Yaskawa INFORM job: kufsa_test_with_table.JBI

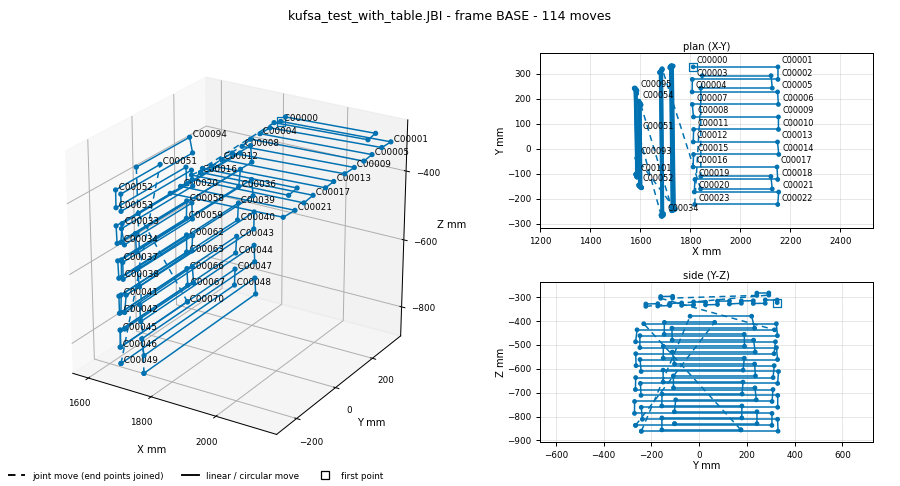
[picture p0: tool path of kufsa_test_with_table.JBI in frame BASE, 114 of 114 moves have a stored position in this frame; points joined in program order, loops and branches not executed]
/JOB
//NAME kufsa_with_table
//POS
///NPOS 114,0,114,0,0,0
///TOOL 0
///POSTYPE BASE
///RECTAN
///RCONF 1,0,0,0,0,0,0,0,0,0,0,0,0,0,0,0,0,0,0,0,0,0,0,0
C00000=1812.070007,326.956462,-322.467041,180.000000,-89.999999,0.000000
C00001=2150.695598,326.956462,-312.028718,180.000000,-89.999999,0.000000
C00002=2150.727599,276.956462,-311.505303,180.000000,-89.999999,0.000000
C00003=1808.470333,276.956462,-325.644002,180.000000,-89.999999,0.000000
C00004=1807.754534,226.956462,-326.266171,180.000000,-89.999999,0.000000
C00005=2149.229584,226.956462,-314.850962,180.000000,-89.999999,0.000000
C00006=2152.427886,176.956462,-315.522758,180.000000,-89.999999,0.000000
C00007=1808.354706,176.956462,-325.499784,180.000000,-89.999999,0.000000
C00008=1813.127705,126.956462,-328.391472,180.000000,-89.999999,0.000000
C00009=2152.547136,126.956462,-316.102628,180.000000,-89.999999,0.000000
C00010=2152.688424,76.956462,-316.428035,180.000000,-89.999999,0.000000
C00011=1813.792182,76.956462,-330.537424,180.000000,-89.999999,0.000000
C00012=1812.079517,26.956462,-332.110167,180.000000,-89.999999,0.000000
C00013=2148.963612,26.956462,-320.940761,180.000000,-89.999999,0.000000
C00014=2153.965148,-23.043538,-319.751379,180.000000,-89.999999,0.000000
C00015=1813.274428,-23.043538,-332.397937,180.000000,-89.999999,0.000000
C00016=1811.443268,-73.043538,-334.200996,180.000000,-89.999999,0.000000
C00017=2146.917653,-73.043538,-323.945193,180.000000,-89.999999,0.000000
C00018=2149.737979,-123.043538,-326.004047,180.000000,-89.999999,0.000000
C00019=1819.062406,-123.043538,-334.939239,180.000000,-89.999999,0.000000
C00020=1816.212947,-173.043538,-337.150638,180.000000,-89.999999,0.000000
C00021=2153.683780,-173.043538,-327.184770,180.000000,-89.999999,0.000000
C00022=2149.816473,-223.043538,-328.439434,180.000000,-89.999999,0.000000
C00023=1817.967726,-223.043538,-338.250259,180.000000,-89.999999,0.000000
C00024=1847.834252,291.859988,-291.167343,180.000000,-89.999999,0.000000
C00025=2123.193751,291.859988,-282.202509,180.000000,-89.999999,0.000000
C00026=2127.968562,241.859988,-282.721095,180.000000,-89.999999,0.000000
C00027=1842.147711,241.859988,-292.609524,180.000000,-89.999999,0.000000
C00028=1842.355615,-110.851952,-303.697098,180.000000,-89.999999,0.000000
C00029=2122.511360,-110.851952,-296.331318,180.000000,-89.999999,0.000000
C00030=2127.898871,-160.851952,-297.180806,180.000000,-89.999999,0.000000
C00031=1841.572191,-160.851952,-304.679312,180.000000,-89.999999,0.000000
C00032=1689.025256,316.314359,-436.599221,180.000000,-89.999999,0.000000
C00033=1693.340579,-259.742111,-436.599221,180.000000,-89.999999,0.000000
C00034=1692.565910,-265.923822,-486.599221,180.000000,-89.999999,0.000000
C00035=1687.558336,319.676130,-486.599221,180.000000,-89.999999,0.000000
C00036=1685.839030,313.772706,-536.599221,180.000000,-89.999999,0.000000
C00037=1691.883319,-265.207335,-536.599221,180.000000,-89.999999,0.000000
C00038=1690.585462,-264.079002,-586.599221,180.000000,-89.999999,0.000000
C00039=1684.578004,314.403429,-586.599221,180.000000,-89.999999,0.000000
C00040=1684.322900,309.849895,-636.599221,180.000000,-89.999999,0.000000
C00041=1689.091070,-265.469540,-636.599221,180.000000,-89.999999,0.000000
C00042=1687.752456,-266.658623,-686.599221,180.000000,-89.999999,0.000000
C00043=1681.655032,309.368812,-686.599221,180.000000,-89.999999,0.000000
C00044=1680.951913,305.521491,-736.599221,180.000000,-89.999999,0.000000
C00045=1687.427916,-270.100352,-736.599221,180.000000,-89.999999,0.000000
C00046=1685.190554,-270.446758,-786.599221,180.000000,-89.999999,0.000000
C00047=1678.938861,305.219084,-786.599221,180.000000,-89.999999,0.000000
C00048=1677.146797,304.775970,-836.599221,180.000000,-89.999999,0.000000
C00049=1683.692237,-266.007352,-836.599221,180.000000,-89.999999,0.000000
C00050=1683.692237,-266.007352,-836.599221,180.000000,-89.999999,0.000000
C00051=1592.682564,65.013086,-405.440930,180.000000,-89.999999,0.000000
C00052=1593.996273,-145.301390,-405.440930,180.000000,-89.999999,0.000000
C00053=1594.466635,-146.306407,-455.440930,180.000000,-89.999999,0.000000
C00054=1593.576386,188.991519,-455.440930,180.000000,-89.999999,0.000000
C00055=1594.547485,190.175259,-505.440930,180.000000,-89.999999,0.000000
C00056=1596.012621,-149.877854,-505.440930,180.000000,-89.999999,0.000000
C00057=1598.057111,-150.260962,-555.440930,180.000000,-89.999999,0.000000
C00058=1594.819072,189.154091,-555.440930,180.000000,-89.999999,0.000000
C00059=1596.462882,184.159348,-605.440930,180.000000,-89.999999,0.000000
C00060=1599.097893,-150.679694,-605.440930,180.000000,-89.999999,0.000000
C00061=1601.194645,-150.579766,-655.440930,180.000000,-89.999999,0.000000
C00062=1596.716601,183.692011,-655.440930,180.000000,-89.999999,0.000000
C00063=1598.777618,180.083430,-705.440930,180.000000,-89.999999,0.000000
C00064=1603.311051,-155.279706,-705.440930,180.000000,-89.999999,0.000000
C00065=1604.512194,-156.238230,-755.440930,180.000000,-89.999999,0.000000
C00066=1599.772168,179.164152,-755.440930,180.000000,-89.999999,0.000000
C00067=1602.114821,178.707079,-805.440930,180.000000,-89.999999,0.000000
C00068=1604.713204,-155.716551,-805.440930,180.000000,-89.999999,0.000000
C00069=1606.157345,-155.900105,-855.440930,180.000000,-89.999999,0.000000
C00070=1603.002390,174.947550,-855.440930,180.000000,-89.999999,0.000000
C00071=1603.002390,174.947550,-855.440930,180.000000,-89.999999,0.000000
C00072=1724.578416,-231.807524,-411.083672,180.000000,-89.999999,0.000000
C00073=1718.279325,323.447595,-411.083672,180.000000,-89.999999,0.000000
C00074=1719.725414,327.955120,-461.083672,180.000000,-89.999999,0.000000
C00075=1725.796875,-247.885600,-461.083672,180.000000,-89.999999,0.000000
C00076=1727.476934,-248.031667,-511.083672,180.000000,-89.999999,0.000000
C00077=1721.770468,323.709354,-511.083672,180.000000,-89.999999,0.000000
C00078=1723.614458,328.610857,-561.083672,180.000000,-89.999999,0.000000
C00079=1728.674863,-247.324114,-561.083672,180.000000,-89.999999,0.000000
C00080=1731.265446,-242.598605,-611.083672,180.000000,-89.999999,0.000000
C00081=1724.878351,332.404799,-611.083672,180.000000,-89.999999,0.000000
C00082=1725.967145,328.907011,-661.083672,180.000000,-89.999999,0.000000
C00083=1733.123323,-245.670029,-661.083672,180.000000,-89.999999,0.000000
C00084=1733.584924,-243.188232,-711.083672,180.000000,-89.999999,0.000000
C00085=1726.804307,329.270615,-711.083672,180.000000,-89.999999,0.000000
C00086=1729.229751,328.994115,-761.083672,180.000000,-89.999999,0.000000
C00087=1734.901952,-242.222270,-761.083672,180.000000,-89.999999,0.000000
C00088=1737.913833,-237.463930,-811.083672,180.000000,-89.999999,0.000000
C00089=1730.236277,328.580483,-811.083672,180.000000,-89.999999,0.000000
C00090=1731.867128,330.516874,-861.083672,180.000000,-89.999999,0.000000
C00091=1739.462265,-241.828515,-861.083672,180.000000,-89.999999,0.000000
C00092=1739.462265,-241.828515,-861.083672,180.000000,-89.999999,0.000000
C00093=1586.192316,-37.777443,-379.657788,180.000000,-89.999999,0.000000
C00094=1586.018778,220.048604,-379.657788,180.000000,-89.999999,0.000000
C00095=1587.115619,232.433194,-429.657788,180.000000,-89.999999,0.000000
C00096=1587.946012,-113.769722,-429.657788,180.000000,-89.999999,0.000000
C00097=1586.574680,-112.699043,-479.657788,180.000000,-89.999999,0.000000
C00098=1585.601795,228.117871,-479.657788,180.000000,-89.999999,0.000000
C00099=1584.980452,234.981511,-529.657788,180.000000,-89.999999,0.000000
C00100=1586.351337,-112.328011,-529.657788,180.000000,-89.999999,0.000000
C00101=1587.981300,-102.830919,-579.657788,180.000000,-89.999999,0.000000
C00102=1583.294206,232.360436,-579.657788,180.000000,-89.999999,0.000000
C00103=1582.141752,235.917997,-629.657788,180.000000,-89.999999,0.000000
C00104=1584.825898,-107.857211,-629.657788,180.000000,-89.999999,0.000000
C00105=1584.372957,-107.195150,-679.657788,180.000000,-89.999999,0.000000
C00106=1583.512190,233.854829,-679.657788,180.000000,-89.999999,0.000000
C00107=1577.236228,239.550729,-729.657788,180.000000,-89.999999,0.000000
C00108=1586.464349,-97.948331,-729.657788,180.000000,-89.999999,0.000000
C00109=1584.137106,-103.589890,-779.657788,180.000000,-89.999999,0.000000
C00110=1576.249941,242.210446,-779.657788,180.000000,-89.999999,0.000000
C00111=1580.180793,242.276562,-829.657788,180.000000,-89.999999,0.000000
C00112=1582.279332,-102.714387,-829.657788,180.000000,-89.999999,0.000000
C00113=1582.279332,-102.714387,-829.657788,180.000000,-89.999999,0.000000
///POSTYPE PULSE
///PULSE
EC00000=0
EC00001=0
EC00002=0
EC00003=0
EC00004=0
EC00005=0
EC00006=0
EC00007=0
EC00008=0
EC00009=0
EC00010=0
EC00011=0
EC00012=0
EC00013=0
EC00014=0
EC00015=0
EC00016=0
EC00017=0
EC00018=0
EC00019=0
EC00020=0
EC00021=0
EC00022=0
EC00023=0
EC00024=0
EC00025=0
EC00026=0
EC00027=0
EC00028=0
EC00029=0
EC00030=0
EC00031=0
EC00032=0
EC00033=0
EC00034=0
EC00035=0
EC00036=0
EC00037=0
EC00038=0
EC00039=0
EC00040=0
EC00041=0
EC00042=0
EC00043=0
EC00044=0
EC00045=0
EC00046=0
EC00047=0
EC00048=0
EC00049=0
EC00050=92160
EC00051=92160
EC00052=92160
EC00053=92160
EC00054=92160
EC00055=92160
EC00056=92160
EC00057=92160
EC00058=92160
EC00059=92160
EC00060=92160
EC00061=92160
EC00062=92160
EC00063=92160
EC00064=92160
EC00065=92160
EC00066=92160
EC00067=92160
EC00068=92160
EC00069=92160
EC00070=92160
EC00071=184320
EC00072=184320
EC00073=184320
EC00074=184320
EC00075=184320
EC00076=184320
EC00077=184320
EC00078=184320
EC00079=184320
EC00080=184320
EC00081=184320
EC00082=184320
EC00083=184320
EC00084=184320
EC00085=184320
EC00086=184320
EC00087=184320
EC00088=184320
EC00089=184320
EC00090=184320
EC00091=184320
EC00092=276480
EC00093=276480
EC00094=276480
EC00095=276480
EC00096=276480
EC00097=276480
EC00098=276480
EC00099=276480
EC00100=276480
EC00101=276480
EC00102=276480
EC00103=276480
EC00104=276480
EC00105=276480
EC00106=276480
EC00107=276480
EC00108=276480
EC00109=276480
EC00110=276480
EC00111=276480
EC00112=276480
EC00113=368640
//INST
///DATE 2023/01/16 14:01
///ATTR SC,RW,RJ
////FRAME BASE
///GROUP1 RB1,ST1
NOP
MOVJ C00000 EC00000 VJ=15.0
CALL JOB:SPYON
MOVL C00001 EC00001 V=200.0
MOVL C00002 EC00002 V=200.0
MOVL C00003 EC00003 V=200.0
MOVL C00004 EC00004 V=200.0
MOVL C00005 EC00005 V=200.0
MOVL C00006 EC00006 V=200.0
MOVL C00007 EC00007 V=200.0
MOVL C00008 EC00008 V=200.0
MOVL C00009 EC00009 V=200.0
MOVL C00010 EC00010 V=200.0
MOVL C00011 EC00011 V=200.0
MOVL C00012 EC00012 V=200.0
MOVL C00013 EC00013 V=200.0
MOVL C00014 EC00014 V=200.0
MOVL C00015 EC00015 V=200.0
MOVL C00016 EC00016 V=200.0
MOVL C00017 EC00017 V=200.0
MOVL C00018 EC00018 V=200.0
MOVL C00019 EC00019 V=200.0
MOVL C00020 EC00020 V=200.0
MOVL C00021 EC00021 V=200.0
MOVL C00022 EC00022 V=200.0
MOVL C00023 EC00023 V=200.0
CALL JOB:SPYOF
MOVJ C00024 EC00024 VJ=15.0
CALL JOB:SPYON
MOVL C00025 EC00025 V=200.0
MOVL C00026 EC00026 V=200.0
MOVL C00027 EC00027 V=200.0
CALL JOB:SPYOF
MOVJ C00028 EC00028 VJ=15.0
CALL JOB:SPYON
MOVL C00029 EC00029 V=200.0
MOVL C00030 EC00030 V=200.0
MOVL C00031 EC00031 V=200.0
CALL JOB:SPYOF
CALL JOB:GO_HOME
MOVJ C00032 EC00032 VJ=15.0
CALL JOB:SPYON
MOVL C00033 EC00033 V=200.0
MOVL C00034 EC00034 V=200.0
MOVL C00035 EC00035 V=200.0
MOVL C00036 EC00036 V=200.0
MOVL C00037 EC00037 V=200.0
MOVL C00038 EC00038 V=200.0
MOVL C00039 EC00039 V=200.0
MOVL C00040 EC00040 V=200.0
MOVL C00041 EC00041 V=200.0
MOVL C00042 EC00042 V=200.0
MOVL C00043 EC00043 V=200.0
MOVL C00044 EC00044 V=200.0
MOVL C00045 EC00045 V=200.0
MOVL C00046 EC00046 V=200.0
MOVL C00047 EC00047 V=200.0
MOVL C00048 EC00048 V=200.0
MOVL C00049 EC00049 V=200.0
CALL JOB:SPYOF
CALL JOB:GO_HOME
MOVL C00050 EC00050 V=200.0
MOVJ C00051 EC00051 VJ=15.0
CALL JOB:SPYON
MOVL C00052 EC00052 V=200.0
MOVL C00053 EC00053 V=200.0
MOVL C00054 EC00054 V=200.0
MOVL C00055 EC00055 V=200.0
MOVL C00056 EC00056 V=200.0
MOVL C00057 EC00057 V=200.0
MOVL C00058 EC00058 V=200.0
MOVL C00059 EC00059 V=200.0
MOVL C00060 EC00060 V=200.0
MOVL C00061 EC00061 V=200.0
MOVL C00062 EC00062 V=200.0
MOVL C00063 EC00063 V=200.0
MOVL C00064 EC00064 V=200.0
MOVL C00065 EC00065 V=200.0
MOVL C00066 EC00066 V=200.0
MOVL C00067 EC00067 V=200.0
MOVL C00068 EC00068 V=200.0
MOVL C00069 EC00069 V=200.0
MOVL C00070 EC00070 V=200.0
CALL JOB:SPYOF
CALL JOB:GO_HOME
MOVL C00071 EC00071 V=200.0
MOVJ C00072 EC00072 VJ=15.0
CALL JOB:SPYON
MOVL C00073 EC00073 V=200.0
MOVL C00074 EC00074 V=200.0
MOVL C00075 EC00075 V=200.0
MOVL C00076 EC00076 V=200.0
MOVL C00077 EC00077 V=200.0
MOVL C00078 EC00078 V=200.0
MOVL C00079 EC00079 V=200.0
MOVL C00080 EC00080 V=200.0
MOVL C00081 EC00081 V=200.0
MOVL C00082 EC00082 V=200.0
MOVL C00083 EC00083 V=200.0
MOVL C00084 EC00084 V=200.0
MOVL C00085 EC00085 V=200.0
MOVL C00086 EC00086 V=200.0
MOVL C00087 EC00087 V=200.0
MOVL C00088 EC00088 V=200.0
MOVL C00089 EC00089 V=200.0
MOVL C00090 EC00090 V=200.0
MOVL C00091 EC00091 V=200.0
CALL JOB:SPYOF
CALL JOB:GO_HOME
MOVL C00092 EC00092 V=200.0
MOVJ C00093 EC00093 VJ=15.0
CALL JOB:SPYON
MOVL C00094 EC00094 V=200.0
MOVL C00095 EC00095 V=200.0
MOVL C00096 EC00096 V=200.0
MOVL C00097 EC00097 V=200.0
MOVL C00098 EC00098 V=200.0
MOVL C00099 EC00099 V=200.0
MOVL C00100 EC00100 V=200.0
MOVL C00101 EC00101 V=200.0
MOVL C00102 EC00102 V=200.0
MOVL C00103 EC00103 V=200.0
MOVL C00104 EC00104 V=200.0
MOVL C00105 EC00105 V=200.0
MOVL C00106 EC00106 V=200.0
MOVL C00107 EC00107 V=200.0
MOVL C00108 EC00108 V=200.0
MOVL C00109 EC00109 V=200.0
MOVL C00110 EC00110 V=200.0
MOVL C00111 EC00111 V=200.0
MOVL C00112 EC00112 V=200.0
CALL JOB:SPYOF
CALL JOB:GO_HOME
MOVL C00113 EC00113 V=200.0
END
